FUNCTION_BLOCK MultiAgentSystem (* JADE WORKER *)
  (* Standard: 61499-1 *)
  (* Version 1.0, 2014-04-22, Ahmed, Fraunhofer IGD *)
  (* Compiler header: package fb.rt; *)
  (* Compiler Java Sun JDK 1.5.0 *)
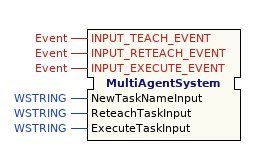
  EVENT_INPUT
    INPUT_TEACH_EVENT;
    INPUT_RETEACH_EVENT;
    INPUT_EXECUTE_EVENT;
  END_EVENT
  VAR_INPUT
    NewTaskNameInput : WSTRING;
    ReteachTaskInput : WSTRING;
    ExecuteTaskInput : WSTRING;
  END_VAR
END_FUNCTION_BLOCK
